TYPE
PLCopenCommandGroupInternal:
STRUCT
  Working : BOOL;
  SubscriberCount : INT;
  Subscriber : ARRAY[0..GVLTcCommando.MAX_RELATED_GROUPS] OF PLCopenRemote;
END_STRUCT
END_TYPE

(* stored: Version 1.1.0.1
   DUT PLCopenCommandGroupInternal: Id {f2eaeac7-e209-40d2-95ee-fa36a7e2cbeb} *)
